lSecondaryPowerSupplyB.Name := 'cSecondaryB';
lSecondaryPowerSupplyB.SubSystem := cSubsystemSecondary;
lSecondaryPowerSupplyB.NetworkId := 1;
lSecondaryPowerSupplyB.initializeSecondary(gSystemPrimary.SecondaryPowerSupply);
registerOperational(ADR(lSecondaryPowerSupplyB));

SUPER^.initialize();
SubSystem := cSubsystemCANBusSystem;

lOperationalSystemStateScope := cSystemStatePreparing;
lAllowableUpSystemStateScope := cSystemStateStandby;
lSystemControlRecovery := cSystemControlReset;	

lBusPower.OutputSystemState := cSystemStateStandby;
lEstopOnNodeState := FALSE;
                
END_METHOD

(* {attribute 'monitoring' := 'call'} *)
PROPERTY SecondaryPowerSupplyB : REFERENCE TO ControllerSecondaryPowerSupply
GET
                    SecondaryPowerSupplyB ref= lSecondaryPowerSupplyB;
                  
END_GET
END_PROPERTY

(* {attribute 'monitoring' := 'call'} *)
PROPERTY SecondaryPowerSupplyA : REFERENCE TO ControllerSecondaryPowerSupply
GET
                    SecondaryPowerSupplyA ref= lSecondaryPowerSupplyA;
                  
END_GET
END_PROPERTY
END_FUNCTION_BLOCK

FUNCTION_BLOCK CyclePrimary EXTENDS Cycle
  VAR
    lVROperationalHours : ValueReferencePersistentReal;
    lOperationalHours : t_persistent_real;
    lVRHours : ValueReferencePersistentReal;
    lHours : t_persistent_real;
    lOperationalHoursMeterTickPrevious : ULINT := 0;
    lOperationalHoursMeterTickPeriod : ULINT := ((1000000 * 60) * 10);
    lOperationalHoursMeterTickOffset : ULINT := ((1000000 * 60) * 5);
    lHoursMeterTickPrevious : ULINT := 0;
    lHoursMeterTickPeriod : ULINT := ((1000000 * 60) * 60);
    lHoursMeterTickOffset : ULINT := ((1000000 * 60) * 30);
  END_VAR

            ;
          

METHOD initialize
                  lVROperationalHours.initializeValueReference(lOperationalHours,NopSelf,'OpHours','Operational hours','',cValueStyleParameter);
lOperationalHours.Identifier := t_persistent_id.cPersistentID_OperationalHours;
lOperationalHours.initialize();

lVRHours.initializeValueReference(lHours,NopSelf,'AllHours','System up-time hours','',cValueStyleParameter);
lHours.Identifier := t_persistent_id.cPersistentID_Hours;
lHours.initialize();

SUPER^.initialize();

lOperationalHoursMeterTickPrevious := lCurrentTime.Value;
lHoursMeterTickPrevious := lCurrentTime.Value;

                
END_METHOD

METHOD operator
                  SUPER^.operator();

IF ((gSystemPrimary.SystemState.State<cSystemStateOperational) AND
	(lCurrentTime.Value>lOperationalHoursMeterTickOffset)) THEN
	lOperationalHoursMeterTickPrevious := lCurrentTime.Value - lOperationalHoursMeterTickOffset;
END_IF
IF (lCurrentTime.Value > (lOperationalHoursMeterTickPrevious+lOperationalHoursMeterTickPeriod)) THEN
	lOperationalHoursMeterTickPrevious := lOperationalHoursMeterTickPrevious + lOperationalHoursMeterTickPeriod;
	lOperationalHours.Value := lOperationalHours.Value + ULINT_TO_REAL(lOperationalHoursMeterTickPeriod)/3600000000;
END_IF

IF (lCurrentTime.Value>lHoursMeterTickOffset) THEN
	lHoursMeterTickPrevious := lCurrentTime.Value - lHoursMeterTickOffset;
END_IF
IF (lCurrentTime.Value > (lHoursMeterTickPrevious+lHoursMeterTickPeriod)) THEN
	lHoursMeterTickPrevious := lHoursMeterTickPrevious + lHoursMeterTickPeriod;
	lHours.Value := lHours.Value + ULINT_TO_REAL(lHoursMeterTickPeriod)/3600000000;
END_IF



                
END_METHOD

PROPERTY Hours : REAL
GET
                    Hours := lHours.Value;
                  
END_GET
SET
                    lHours.Value := Hours;
                  
END_SET
END_PROPERTY

PROPERTY OperationalHours : REAL
GET
                    OperationalHours := lOperationalHours.Value;
                  
END_GET
SET
                    lOperationalHours.Value := OperationalHours;
                  
END_SET
END_PROPERTY

PROPERTY TriggerResetHours : BOOL
SET
                    IF (TriggerResetHours) THEN
	lHours.Value := 0.0;
END_IF
                  
END_SET
END_PROPERTY

PROPERTY TriggerResetOperationalHours : BOOL
SET
                    IF (TriggerResetOperationalHours) THEN
	lOperationalHours.Value := 0.0;
END_IF

                  
END_SET
END_PROPERTY
END_FUNCTION_BLOCK

FUNCTION_BLOCK LEDDiagnosticPrimary EXTENDS LEDDiagnostic
  VAR CONSTANT
    cColorRed : UINT := X_SYS_LED_COLOR_RED;
    cColorGreen : UINT := X_SYS_LED_COLOR_GREEN;
    cColorYellow : UINT := X_SYS_LED_COLOR_YELLOW;
    cColorOrange : UINT := X_SYS_LED_COLOR_ORANGE;
  END_VAR
  VAR
    lState : ValueObjectBoolOutputReferenceUSINTAsBool;
    lColor : ValueObjectUINTOutputReferenceUINT;
    lCounter : UINT := 0;
    lTimer : t_timer;
  END_VAR

            
          

METHOD operator
                  CASE lCode OF
	cLEDCodeNone,
	cLEDCodeStartup:
		scrollBidirectional(1);
	
	cLEDCodeNormal:
		flash(T#500MS,T#500MS,cColorGreen);
	
	cLEDCodeStandby:
		scrollUnidirectional(1);
	
	cLEDCodeMaintenance:
		flash(T#500MS,T#500MS,cColorYellow);

	cLEDCodeSoftwareCrash:
		flash(T#500MS,T#500MS,cColorRed);
		
	cLEDCodeWatchDogDisabled:
		flash(T#125MS,T#125MS,cColorGreen);

	cLEDCodeFailSafe:
		flash(T#125MS,T#125MS,cColorYellow);
		
	cLEDCodeFailSafeSevere:
		flash(T#125MS,T#125MS,cColorRed);
END_CASE

SUPER^.operator();


                
END_METHOD

METHOD initialize
                  lState.initializeValueObjectOp(OpSelf,'State','Diagnostic LED pattern','',cValueStyleConfigurable);
lColor.initializeValueObjectOp(OpSelf,'Color','Diagnostic LED color','',cValueStyleConfigurable);

SUPER^.initialize();

lTimer.Enable := TRUE;
lTimer.Period := T#1S;
lTimer.initialize();

                
END_METHOD

METHOD initializeLEDDiagnostic
  VAR_INPUT
    state : REFERENCE TO USINT;
    color : REFERENCE TO UINT;
  END_VAR
                  lState.OutputReference REF= state;
lColor.OutputReference REF= color;

                
END_METHOD

METHOD scrollBidirectional
  VAR_INPUT
    rate : USINT;
  END_VAR
  VAR
    index : UINT;
  END_VAR
                  lCounter := lCounter + 1;
index := lCounter/rate;

IF (index>200) THEN
	lCounter := 0;
	index := 0;
END_IF

IF (index>100) THEN
	lColor.Value := index - 100;
ELSE
	lColor.Value := 100 - index;
END_IF

lState.Value := TRUE;

                
END_METHOD

METHOD scrollUnidirectional
  VAR_INPUT
    rate : USINT;
  END_VAR
  VAR
    index : UINT;
  END_VAR
                  lCounter := lCounter + 1;
index := lCounter/rate;

IF (index>100) THEN
	lCounter := 0;
	index := 0;
END_IF

lColor.Value := index;
lState.Value := TRUE;

                
END_METHOD

METHOD flash
  VAR_INPUT
    off : t_time;
    on : t_time;
    color : UINT;
  END_VAR
                  lTimer.operator();

IF (lTimer.Expired) THEN
	IF (lState.Value) THEN
		lTimer.Period := off;
	ELSE
		lTimer.Period := on;
	END_IF

	lState.Value := NOT(lState.Value);
	lTimer.reset();
END_IF

lColor.Value := color;

                
END_METHOD
END_FUNCTION_BLOCK

FUNCTION_BLOCK LocalMachinePrimary EXTENDS LocalMachine
  VAR
    lVRWheelBase : ValueReferencePersistentReal;
    lWheelBase : t_persistent_real;
    lVRWheelTrack : ValueReferencePersistentReal;
    lWheelTrack : t_persistent_real;
  END_VAR

            
          

METHOD initialize
                  Name := 'Local';

lVRWheelBase.initializeValueReference(lWheelBase,NopSelf,'WheelBase','Machine wheel base','',cValueStyleParameter);
lWheelBase.Identifier := t_persistent_id.cPersistentID_WheelBase;
lWheelBase.initialize();

lVRWheelTrack.initializeValueReference(lWheelTrack,NopSelf,'WheelTrack','Machine wheel track','',cValueStyleParameter);
lWheelTrack.Identifier := t_persistent_id.cPersistentID_WheelTrack;
lWheelTrack.initialize();

SUPER^.initialize();

                
END_METHOD

METHOD defaultPersistence
  VAR
    parameter : t_token_string;
    value : t_token_string;
  END_VAR
                  SUPER^.defaultPersistence();

WheelBase := 5000;
WheelTrack := 4100;

                
END_METHOD

PROPERTY WheelBase : REAL
GET
                    WheelBase := lWheelBase.Value;
                  
END_GET
SET
                    lWheelBase.Value := WheelBase;
                  
END_SET
END_PROPERTY

PROPERTY WheelTrack : REAL
GET
                    WheelTrack := lWheelTrack.Value;
                  
END_GET
SET
                    lWheelTrack.Value := WheelTrack;
                  
END_SET
END_PROPERTY
END_FUNCTION_BLOCK

FUNCTION_BLOCK SystemPrimary EXTENDS System
  VAR CONSTANT
    cOuterRegionSteer : t_percentage := 1.0;
    cInnerRegionSteer : t_percentage := 0.98;
    cInnerValueSteer : t_percentage := 1.0;
    cOuterValueSteer : t_percentage := 0.0;
    cZeroThresholdSteer : t_percentage := 0.03;
  END_VAR
  VAR
    lLEDDiagnostic : LEDDiagnosticPrimary;
    lCycle : CyclePrimary;
    lExecutor : Executor;
    lPLC : PLCPrimary;
    lSystemState : SystemState;
    lParseServerRO : ParseTCPServer;  (* lEchoServer: EchoTCPServer; *)
    lParseServerRW : ParseTCPServer;
    lParseServerEdge : ParseTCPServer;
    lMetric0ms : ParticleReporterEvent;
    lMetric250ms : ParticleReporterEvent;
    lMetric500ms : ParticleReporterEvent;
    lMetric1s : ParticleReporterEvent;
    lMetric5s : ParticleReporterEvent;
    lMetric1m : ParticleReporterEvent;
    lMetric1h : ParticleReporterEvent;
    lMetric1d : ParticleReporterEvent;
    lOperatingMode : OperatingMode;
    lActive : ActiveSystem;
    lUMFS : UMFS;
    lEstopLoad : EstopLoad;
    lTMS : TMS;
    lSecondaryPowerSupply : SecondaryPowerSupplyPrimary;
    lAlarm : Alarm;
    lBeacons : Beacons;
    lHorn : Horn;
    lLights : Lights;
    lSensorSupply : SensorSupply;
    lSteering : SteerMovementElectric;
    lSteerAPositionInterlock : WrapperScaledInterlock;
    lSteerBPositionInterlock : WrapperScaledInterlock;
    lSteerCPositionInterlock : WrapperScaledInterlock;
    lSteerDPositionInterlock : WrapperScaledInterlock;
    _LocalMachinePrimary : REFERENCE TO LocalMachinePrimary;
    _CANOpenMasterSystemPrimary : REFERENCE TO CANOpenMasterSystemPrimary;
    _CANOpenMasterDrivePrimary : REFERENCE TO CANOpenMasterDrivePrimary;
    _UIEvent : REFERENCE TO UIEvent;
    _FunctionalModeControl : REFERENCE TO FunctionalModeControl;
    _UInterface : REFERENCE TO UInterface;
    _BMS : REFERENCE TO BMS;
    _Charger : REFERENCE TO Charger;
    _ProgrammedMovementControl : REFERENCE TO ProgrammedMovementControl;
    _Lift : REFERENCE TO QuadMovement;
    _Travel : REFERENCE TO CheckedMovement;
  END_VAR

            ;
          

METHOD initializeStage2
                  (*registerOperational(ADR(lEchoServer));
lEchoServer.Name := 'EchoTCP:49860';
lEchoServer.ServerPort := 49860;
lEchoServer.ServerPortLower := 49860;
lEchoServer.ServerPortUpper := 49869;*)

registerOperational(ADR(lParseServerRW));
lParseServerRW.Name := 'ParserRW';
lParseServerRW.ServerPort := 49870;
lParseServerRW.ServerPortLower := 49870;
lParseServerRW.ServerPortUpper := 49879;
lParseServerRW.ReadWrite := TRUE;
lParseServerRW.Interactive := TRUE;
lParseServerRW.WrappedResponse := FALSE;
lParseServerRW.ReportError := TRUE;

registerOperational(ADR(lParseServerRO));
lParseServerRO.Name := 'ParserRO';
lParseServerRO.ServerPort := 49880;
lParseServerRO.ServerPortLower := 49880;
lParseServerRO.ServerPortUpper := 49889;
lParseServerRO.ReadWrite := FALSE;
lParseServerRO.Interactive := TRUE;
lParseServerRO.WrappedResponse := FALSE;
lParseServerRO.ReportError := TRUE;

registerOperational(ADR(lParseServerEdge));
lParseServerEdge.Name := 'ParserEdge';
lParseServerEdge.ServerPort := 49860;
lParseServerEdge.ServerPortLower := 49860;
lParseServerEdge.ServerPortUpper := 49869;
lParseServerEdge.ReadWrite := TRUE;
lParseServerEdge.Interactive := FALSE;
lParseServerEdge.WrappedResponse := TRUE;
lParseServerEdge.ReportError := FALSE;

lMetric0ms.Name := 'Metric0ms';
lMetric0ms.initializeEventOp(OpSelf,'',cECMetric);

lMetric250ms.Name := 'Metric250ms';
lMetric250ms.initializeEventOp(OpSelf,'',cECMetric);

lMetric500ms.Name := 'Metric500ms';
lMetric500ms.initializeEventOp(OpSelf,'',cECMetric);

lMetric1s.Name := 'Metric1s';
lMetric1s.initializeEventOp(OpSelf,'',cECMetric);

lMetric5s.Name := 'Metric5s';
lMetric5s.initializeEventOp(OpSelf,'',cECMetric);

lMetric1m.Name := 'Metric1m';
lMetric1m.initializeEventOp(OpSelf,'',cECMetric);

lMetric1h.Name := 'Metric1h';
lMetric1h.initializeEventOp(OpSelf,'',cECMetric);

lMetric1d.Name := 'Metric1d';
lMetric1d.initializeEventOp(OpSelf,'',cECMetric);

SUPER^.initializeStage2();

lMetric0ms.Period := T#0MS;
lMetric250ms.Period := T#250MS;
lMetric500ms.Period := T#500MS;
lMetric1s.Period := T#1S;
lMetric5s.Period := T#5S;
lMetric1m.Period := T#1M;
lMetric1h.Period := T#1H;
lMetric1d.Period := T#1D;

                
END_METHOD

METHOD initializeStage0
                  gNameSpace := 'PrimaryPLC';

IF ((NOT(__ISVALIDREF(gSystemPrimary))) OR
	(NOT(__ISVALIDREF(_LocalMachinePrimary))) OR
	(NOT(__ISVALIDREF(_CANOpenMasterSystemPrimary))) OR
	(NOT(__ISVALIDREF(_CANOpenMasterDrivePrimary))) OR
	(NOT(__ISVALIDREF(_UIEvent))) OR
	(NOT(__ISVALIDREF(_FunctionalModeControl))) OR
	(NOT(__ISVALIDREF(_UInterface))) OR
	(NOT(__ISVALIDREF(_BMS))) OR
	(NOT(__ISVALIDREF(_Charger))) OR
	(NOT(__ISVALIDREF(_ProgrammedMovementControl))) OR
	(NOT(__ISVALIDREF(_Lift))) OR
	(NOT(__ISVALIDREF(_Travel)))) THEN
	gCodeErrorHandler(pMessage:=CONCAT('null reference in ',lIdentity));
END_IF

gSystemServices REF= gSystemPrimary;

_LocalMachine REF= _LocalMachinePrimary;
_LEDDiagnostic REF= lLEDDiagnostic;
_Executor REF= lExecutor;	
_Cycle REF= lCycle;
_PLC REF= lPLC;
_SystemState REF= lSystemState;

registerOperational(ADR(lLEDDiagnostic));

registerOperational(ADR(lExecutor));
lExecutor.Client.ServerPort := 49740;

SUPER^.initializeStage0();
SubSystem := cSubsystemMachine;


                
END_METHOD

METHOD operator
                  SUPER^.operator();

lProceed := TRUE;

                
END_METHOD

METHOD initializeStage1
  VAR
    token : t_token_string;
  END_VAR
                  registerOperational(ADR(lCycle));
registerOperational(ADR(lPLC));
registerOperational(ADR(lSystemState));

SUPER^.initializeStage1();

                
END_METHOD

METHOD initializeStage3
                  registerOperational(ADR(lOperatingMode));
registerOperational(ADR(lActive));
registerOperational(ADR(lUMFS));
lUMFS.lEnableSlave := TRUE;
registerOperational(ADR(lEstopLoad));

registerOperational(ADR(lTMS));
registerOperational(ADR(lSecondaryPowerSupply));

registerOperational(ADR(lAlarm));
registerOperational(ADR(lBeacons));
registerOperational(ADR(lHorn));
registerOperational(ADR(lLights));
registerOperational(ADR(lSensorSupply));

registerOperational(ADR(lSteering));

lSteerAPositionInterlock.Name := 'iSteerAPos';
lSteerAPositionInterlock.Input REF= gSystemPrimary.CANOpenMasterDrivePrimary.SteerAngleA.PositionObject;
lSteerAPositionInterlock.Transform.InnerRegion := cInnerRegionSteer;
lSteerAPositionInterlock.Transform.OuterRegion := cOuterRegionSteer;
lSteerAPositionInterlock.Transform.InnerValue := cInnerValueSteer;
lSteerAPositionInterlock.Transform.OuterValue := cOuterValueSteer;
lSteerAPositionInterlock.Client.registerServer(gSystemPrimary.Steering.WheelA.Interlock);
lSteerAPositionInterlock.Client.ScalingContext REF= gSystemPrimary.Steering.WheelA.InputObject;
lSteerAPositionInterlock.Client.ZeroThreshold := cZeroThresholdSteer;
lSteerAPositionInterlock.Sign := -1.0;
lSteerAPositionInterlock.SubSystem := cSubsystemSteerA;
registerOperational(ADR(lSteerAPositionInterlock));

lSteerBPositionInterlock.Name := 'iSteerBPos';
lSteerBPositionInterlock.Input REF= gSystemPrimary.CANOpenMasterDrivePrimary.SteerAngleB.PositionObject;
lSteerBPositionInterlock.Transform.InnerRegion := cInnerRegionSteer;
lSteerBPositionInterlock.Transform.OuterRegion := cOuterRegionSteer;
lSteerBPositionInterlock.Transform.InnerValue := cInnerValueSteer;
lSteerBPositionInterlock.Transform.OuterValue := cOuterValueSteer;
lSteerBPositionInterlock.Client.registerServer(gSystemPrimary.Steering.WheelB.Interlock);
lSteerBPositionInterlock.Client.ScalingContext REF= gSystemPrimary.Steering.WheelB.InputObject;
lSteerBPositionInterlock.Client.ZeroThreshold := cZeroThresholdSteer;
lSteerBPositionInterlock.Sign := -1.0;
lSteerBPositionInterlock.SubSystem := cSubsystemSteerB;
registerOperational(ADR(lSteerBPositionInterlock));

lSteerCPositionInterlock.Name := 'iSteerCPos';
lSteerCPositionInterlock.Input REF= gSystemPrimary.CANOpenMasterDrivePrimary.SteerAngleC.PositionObject;
lSteerCPositionInterlock.Transform.InnerRegion := cInnerRegionSteer;
lSteerCPositionInterlock.Transform.OuterRegion := cOuterRegionSteer;
lSteerCPositionInterlock.Transform.InnerValue := cInnerValueSteer;
lSteerCPositionInterlock.Transform.OuterValue := cOuterValueSteer;
lSteerCPositionInterlock.Client.registerServer(gSystemPrimary.Steering.WheelC.Interlock);
lSteerCPositionInterlock.Client.ScalingContext REF= gSystemPrimary.Steering.WheelC.InputObject;
lSteerCPositionInterlock.Client.ZeroThreshold := cZeroThresholdSteer;
lSteerCPositionInterlock.Sign := -1.0;
lSteerCPositionInterlock.SubSystem := cSubsystemSteerC;
registerOperational(ADR(lSteerCPositionInterlock));

lSteerDPositionInterlock.Name := 'iSteerDPos';
lSteerDPositionInterlock.Input REF= gSystemPrimary.CANOpenMasterDrivePrimary.SteerAngleD.PositionObject;
lSteerDPositionInterlock.Transform.InnerRegion := cInnerRegionSteer;
lSteerDPositionInterlock.Transform.OuterRegion := cOuterRegionSteer;
lSteerDPositionInterlock.Transform.InnerValue := cInnerValueSteer;
lSteerDPositionInterlock.Transform.OuterValue := cOuterValueSteer;
lSteerDPositionInterlock.Client.registerServer(gSystemPrimary.Steering.WheelD.Interlock);
lSteerDPositionInterlock.Client.ScalingContext REF= gSystemPrimary.Steering.WheelD.InputObject;
lSteerDPositionInterlock.Client.ZeroThreshold := cZeroThresholdSteer;
lSteerDPositionInterlock.Sign := -1.0;
lSteerDPositionInterlock.SubSystem := cSubsystemSteerD;
registerOperational(ADR(lSteerDPositionInterlock));

SUPER^.initializeStage3();

                
END_METHOD

PROPERTY BMS : REFERENCE TO BMS
GET
                    BMS ref= _BMS;
                  
END_GET
END_PROPERTY

PROPERTY Lift : REFERENCE TO QuadMovement
GET
                    Lift ref= _Lift;
                  
END_GET
END_PROPERTY

PROPERTY CANOpenMasterDrivePrimary : REFERENCE TO CANOpenMasterDrivePrimary
GET
                    CANOpenMasterDrivePrimary ref= _CANOpenMasterDrivePrimary;
                  
END_GET
END_PROPERTY

PROPERTY CANOpenMasterSystemPrimary : REFERENCE TO CANOpenMasterSystemPrimary
GET
                    CANOpenMasterSystemPrimary ref= _CANOpenMasterSystemPrimary;
                  
END_GET
END_PROPERTY

PROPERTY Steering : REFERENCE TO SteerMovement
GET
                    Steering ref= lSteering;
                  
END_GET
END_PROPERTY

PROPERTY UInterface : REFERENCE TO UInterface
GET
                    UInterface ref= _UInterface;
                  
END_GET
END_PROPERTY

PROPERTY Travel : REFERENCE TO CheckedMovement
GET
                    Travel ref= _Travel;
                  
END_GET
END_PROPERTY

PROPERTY UIEvent : REFERENCE TO UIEvent
GET
                    UIEvent ref= _UIEvent;
                  
END_GET
END_PROPERTY

PROPERTY FunctionalModeControl : REFERENCE TO FunctionalModeControl
GET
                    FunctionalModeControl ref= _FunctionalModeControl;
                  
END_GET
END_PROPERTY

PROPERTY Active : REFERENCE TO ActiveSystem
GET
                    Active ref= lActive;
                  
END_GET
END_PROPERTY

PROPERTY Lights : REFERENCE TO Lights
GET
                    Lights ref= lLights;
                  
END_GET
END_PROPERTY

PROPERTY OperatingMode : REFERENCE TO OperatingMode
GET
                    OperatingMode ref= lOperatingMode;
                  
END_GET
END_PROPERTY

PROPERTY SecondaryPowerSupply : REFERENCE TO SecondaryPowerSupply
GET
                    SecondaryPowerSupply ref= lSecondaryPowerSupply;
                  
END_GET
END_PROPERTY

PROPERTY LocalMachinePrimary : REFERENCE TO LocalMachinePrimary
GET
                    LocalMachinePrimary ref= _LocalMachinePrimary;
                  
END_GET
END_PROPERTY

PROPERTY ProgrammedMovementControl : REFERENCE TO ProgrammedMovementControl
GET
                    ProgrammedMovementControl ref= _ProgrammedMovementControl;
                  
END_GET
END_PROPERTY

PROPERTY Charger : REFERENCE TO Charger
GET
                    Charger ref= _Charger;
                  
END_GET
END_PROPERTY
END_FUNCTION_BLOCK
